TEXTLIST PrzyciskAlarmy
  1 = 'AKTYWNE'
  0 = 'WSZYSTKIE'
   = ''
END_TEXTLIST

(* stored: Version 1.1.0.1, ProductVersion 3.1.4024.3
   TextList PrzyciskAlarmy: Id {1afdc16d-7865-4c41-89bd-947752b0b602} *)
